PROGRAM MAIN
VAR
	MyAnalogueTerminal : AnalogueTerminal;
END_VAR

END_PROGRAM

(* stored: Version 1.1.0.1, ProductVersion 3.1.4024.12
   POU MAIN: Id {3c71bcc5-3027-453b-a942-efad1d7940d1}, SpecialFunc None *)
